// Mitsubishi GX Works2 project: 서보4   PLC: Q02/Q02H

PROGRAM MAIN
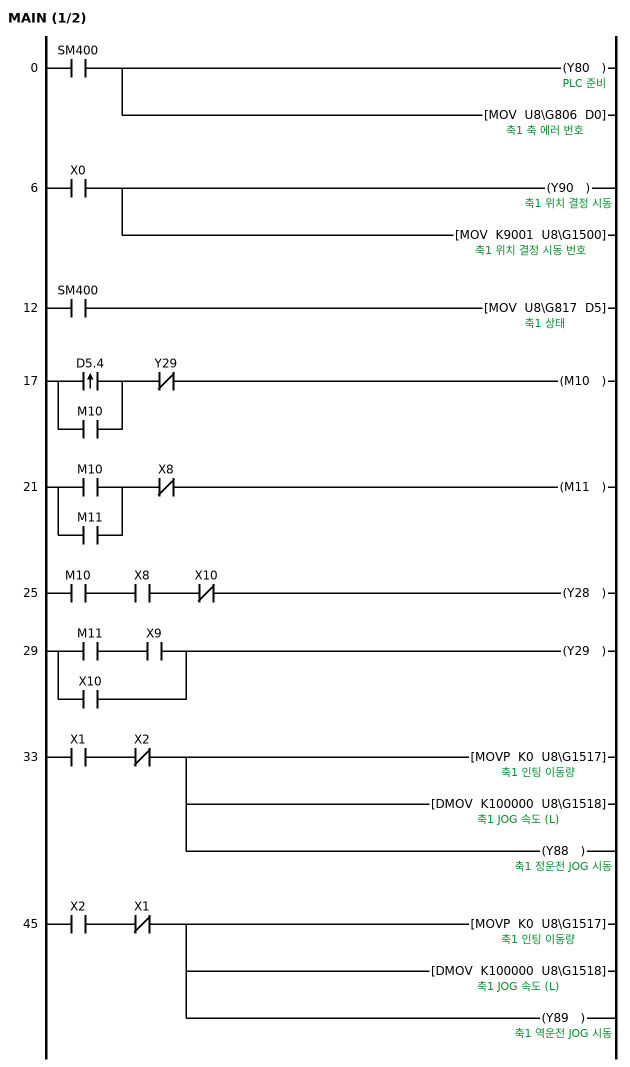
0     LD      SM400
      OUT     Y80  ; PLC 준비
      MOV     U8\G806 D0  ; 축1 축 에러 번호
6     LD      X0
      OUT     Y90  ; 축1 위치 결정 시동
      MOV     K9001 U8\G1500  ; 축1 위치 결정 시동 번호
12    LD      SM400
      MOV     U8\G817 D5  ; 축1 상태
17    LDP     D5.4
      OR      M10
      ANI     Y29
      OUT     M10
21    LD      M10
      OR      M11
      ANI     X8
      OUT     M11
25    LD      M10
      AND     X8
      ANI     X10
      OUT     Y28
29    LD      M11
      AND     X9
      OR      X10
      OUT     Y29
33    LD      X1
      ANI     X2
      MOVP    K0 U8\G1517  ; 축1 인팅 이동량
      DMOV    K100000 U8\G1518  ; 축1 JOG 속도 (L)
      OUT     Y88  ; 축1 정운전 JOG 시동
45    LD      X2
      ANI     X1
      MOVP    K0 U8\G1517
      DMOV    K100000 U8\G1518
      OUT     Y89  ; 축1 역운전 JOG 시동
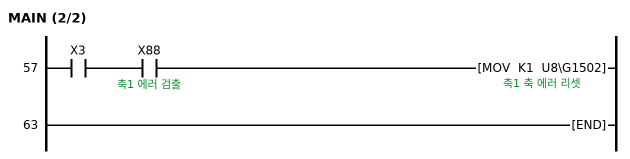
57    LD      X3
      AND     X88  ; 축1 에러 검출
      MOV     K1 U8\G1502  ; 축1 축 에러 리셋
63    END
END_PROGRAM

// device comments not shown above
X80  ; QD75 준비 완료
X81  ; 동기용 플래그
X84  ; 축1 M 코드 ON
X85  ; 축2 M 코드 ON
X89  ; 축2 에러 검출
X8C  ; 축1 BUSY
X8D  ; 축2 BUSY
X90  ; 축1 시동 완료
X91  ; 축2 시동 완료
X94  ; 축1 위치 결정 완료
X95  ; 축2 위치 결정 완료
Y84  ; 축1 축 정지
Y85  ; 축2 축 정지
Y8A  ; 축2 정운전 JOG 시동
Y8B  ; 축2 역운전 JOG 시동
Y91  ; 축2 위치 결정 시동
Y94  ; 축1 실행 금지 플래그
Y95  ; 축2 실행 금지 플래그
